// TIA Portal V18 export
DATA_BLOCK "V90Servo_DB"   // DB2500
VERSION : 0.1
// stored: AutoNumber false, DBAccessibleFromOPCUA true, DBAccessibleFromWebserver true, InstanceOfName V90_Servo, InstanceOfType FB
"V90_Servo"
   // VAR
   //    Servo_380A1 { S7_SetPoint := 'True'} : "fbV90Ctrl";
   //    Servo_381A1 { S7_SetPoint := 'True'} : "fbV90Ctrl";
   //    Servo_382A1 { S7_SetPoint := 'True'} : "fbV90Ctrl";
   //    Servo_383A1 { S7_SetPoint := 'True'} : "fbV90Ctrl";
   //    Servo1 { S7_SetPoint := 'True'} : "SevroStart&PosCheck";
   //    Servo2 { S7_SetPoint := 'True'} : "SevroStart&PosCheck";
   //    Servo3 { S7_SetPoint := 'True'} : "SevroStart&PosCheck";
   //    Servo4 { S7_SetPoint := 'True'} : "SevroStart&PosCheck";
   //    Servo2SafetyPos { S7_SetPoint := 'True'} : DInt;
   //    Servo4SafetyPos { S7_SetPoint := 'True'} : DInt;
   //    IEC_Timer_0_Instance { S7_SetPoint := 'True'} : TON_TIME;
   //    P { S7_SetPoint := 'True'} : Array[0..10] of Bool;
   // END_VAR
BEGIN
END_DATA_BLOCK
